FUNCTION_BLOCK Objet_Pressostat_V1
VAR_INPUT
	Info_Pressostat	:BOOL;	(*nfo détection préssostat / 1 = Détection*)
	Seuil_Press		:REAL;	(*Seuil préssion Réglé sur LE préssostat / en Pa*)
END_VAR
VAR_OUTPUT
END_VAR
VAR
	R_StatDefaut: BOOL;
	R_SeuilPress: REAL;
END_VAR
VAR_IN_OUT
	Tab_Pressostat: Objet_Pressostat;
END_VAR

(* Gestion mesure **************************************************************)
R_StatDefaut	:= Info_Pressostat;
Tab_Pressostat.R_SeuilPress	:= Seuil_Press;

(* Gestion lecture GTC *********************************************************)
Tab_Pressostat.Mot_Lecture.0:= R_StatDefaut;

END_FUNCTION_BLOCK

(* stored: Version 1.1.0.1, ProductVersion 3.1.4024.12
   POU Objet_Pressostat_V1: Id {b7f03509-4d3c-41b0-8e07-2000882081d3}, SpecialFunc None *)
